Fanuc KAREL source: kt00150.KL

-- PROVISIONAL review KL for V1013-1; original PC SHA256 73ebe50e8d074cba1f64d5668e3eca1d8717f766c1e4202b8acabee5fc729c0a
-- Incomplete behavior may be omitted. Consult companion uncertainty JSON. Do not deploy.
PROGRAM KT00150
%NOLOCKGROUP
VAR
  OUT : REAL
-- UNRESOLVED_DECL Y1 type=002018
-- UNRESOLVED_DECL Y2 type=002018
BEGIN
  -- UNRESOLVED_PC offsets 5-19; opcodes 2E,22,9D,33,B2
  -- UNRESOLVED_PC offsets 24-38; opcodes 2E,22,9D,33,B2
  -- UNRESOLVED_PC offsets 43-57; opcodes 2E,22,9D,33,B2
  -- UNRESOLVED_PC offsets 62-76; opcodes 2E,22,9D,33,B2
  -- UNRESOLVED_PC offsets 81-107; opcodes 22,9D,33,B1,22,9D,33,B1,55,64,23
  -- UNRESOLVED_PC offsets 112-116; opcodes 7F
END KT00150
